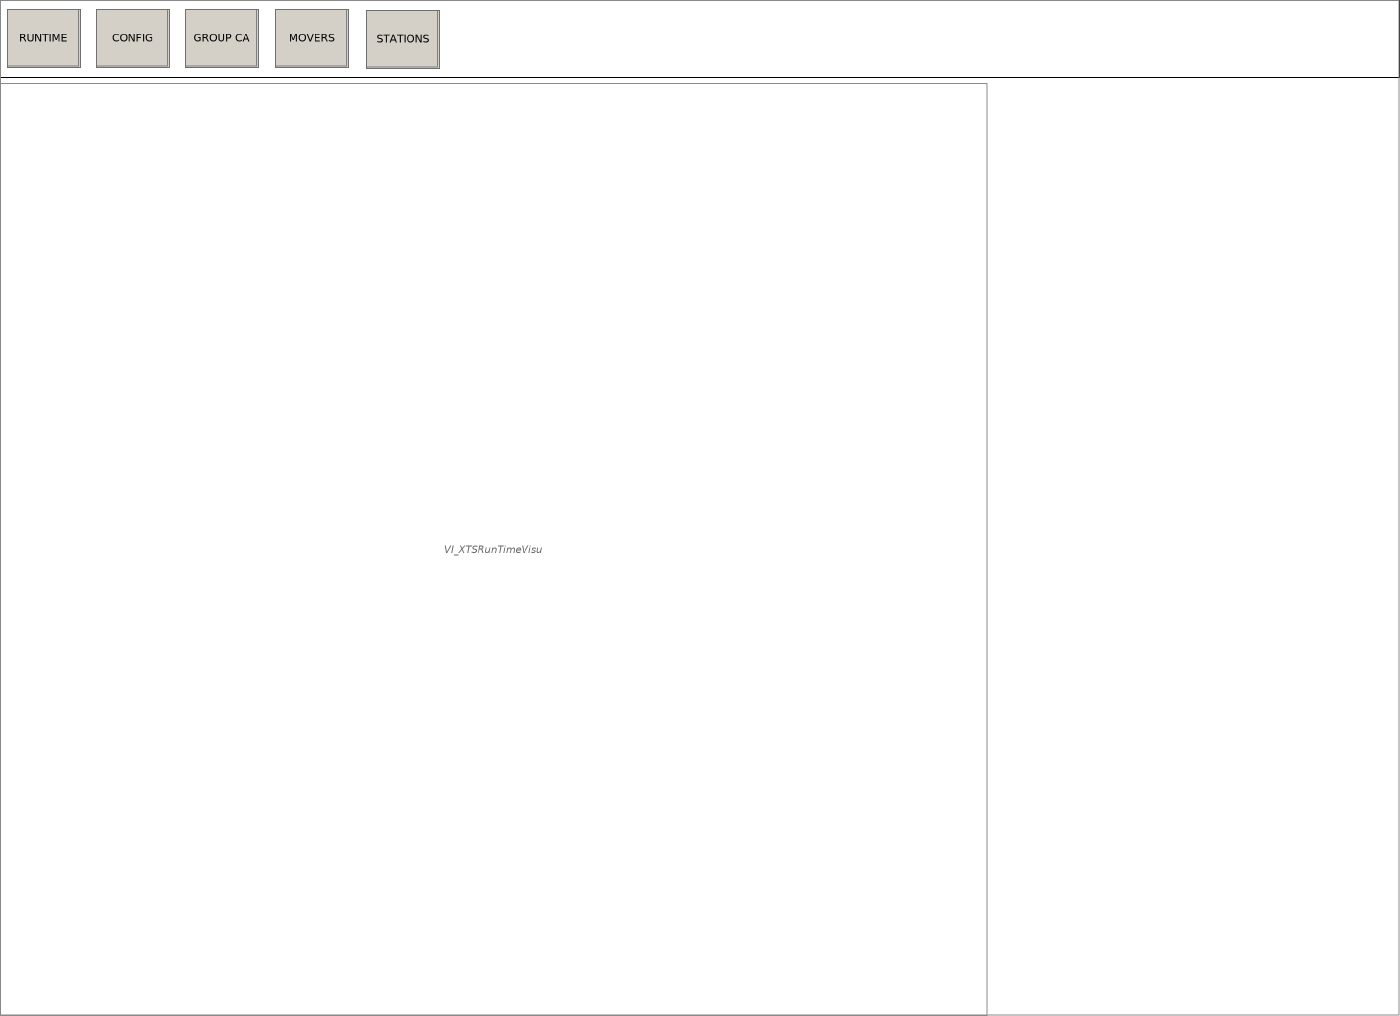
VISUALIZATION VI_XTSMainVisu  // 1430x1038
VAR_IN_OUT
	xts : XTS_System;
END_VAR
    Rectangle (0,0 1430x79)
    Button (7,9 75x60), "RUNTIME", colour toggle: xts.iFrameSelection=0
        OnMouseClick: execute { xts.iFrameSelection := 0; }
    Frame (0,85 1008x953), frame switch variable: xts.iFrameSelection
        shows VI_XTSRunTimeVisu(xts := xts)
        shows VI_XTSConfigurationVisu(xts := xts)
        shows VI_GroupCAVisu(gca := xts.gp)
        shows VI_MoversVisu(ax := xts.ax)
        shows VI_StationsVISU(aStations := xts.aStations)
    Button (98,9 75x60), "CONFIG", colour toggle: xts.iFrameSelection=1
        OnMouseClick: execute { xts.iFrameSelection := 1; }
    Button (189,9 75x60), "GROUP CA", colour toggle: xts.iFrameSelection=2
        OnMouseClick: execute { xts.iFrameSelection := 2; }
    Button (281,9 75x60), "MOVERS", colour toggle: xts.iFrameSelection=3
        OnMouseClick: execute { xts.iFrameSelection := 3; }
    Button (374,10 75x60), "STATIONS", colour toggle: xts.iFrameSelection=4
        OnMouseClick: execute { xts.iFrameSelection := 4; }
END_VISUALIZATION

(* stored: Version 1.1.0.1, ProductVersion 3.1.4024.11
   Visu VI_XTSMainVisu: Id {c4a25e79-daea-4b2a-873a-8fb188555ffe} *)
